FUNCTION_BLOCK fb_ele_io
VAR_IN_OUT
	var_ref_ele : ref_ele_io;
END_VAR
VAR_INPUT
	in_flg_run : BOOL;
	in_wire_sensA : BOOL;
	in_wire_sensB : BOOL;
	in_wire_error : BOOL;
	in_flg_reversal: BOOL;
	in_var_timeout : TIME;
END_VAR
VAR_OUTPUT
	out_flg_run : BOOL;
	out_wire_eleA : BOOL;
	out_wire_eleB : BOOL;
	out_wire_reset : BOOL;

END_VAR
VAR
END_VAR

out_flg_run := in_flg_run;
IF in_flg_reversal THEN
	var_ref_ele.input.in_flg_sensA := in_wire_sensB;
	var_ref_ele.input.in_flg_sensB := in_wire_sensA;
	var_ref_ele.input.in_wire_error := NOT in_wire_error;
	
	out_wire_eleA := var_ref_ele.output.out_flg_eleB;
	out_wire_eleB := var_ref_ele.output.out_flg_eleA;
	out_wire_reset := var_ref_ele.output.out_flg_reset;
ELSE
	var_ref_ele.input.in_flg_sensA := in_wire_sensA;
	var_ref_ele.input.in_flg_sensB := in_wire_sensB;
	var_ref_ele.input.in_wire_error := NOT in_wire_error;
	
	out_wire_eleA := var_ref_ele.output.out_flg_eleA;
	out_wire_eleB := var_ref_ele.output.out_flg_eleB;
	out_wire_reset := var_ref_ele.output.out_flg_reset;
END_IF

IF in_wire_sensA = FALSE AND in_wire_sensB = FALSE THEN
	var_ref_ele.input.in_flg_sensNone := TRUE;
ELSE
	var_ref_ele.input.in_flg_sensNone := FALSE;
END_IF
var_ref_ele.param.var_timeOut := in_var_timeout;

END_FUNCTION_BLOCK

(* stored: Version 1.1.0.1, ProductVersion 3.1.4024.11
   POU fb_ele_io: Id {62fb8b5b-cc73-4fd0-98c9-7e5561bbcfc4}, SpecialFunc None *)
